Fanuc KAREL source: kt00178.KL

-- PROVISIONAL review KL for V1013-1; original PC SHA256 d3c23c733d1c245ba2e05406a3f4e00b66a2d6837c5a015371c1f33c9eca1489
-- Incomplete behavior may be omitted. Consult companion uncertainty JSON. Do not deploy.
PROGRAM KT00178
%NOLOCKGROUP
VAR
  I2 : INTEGER
  OUT : REAL
-- UNRESOLVED_DECL Y1 type=002018
BEGIN
  -- UNRESOLVED_PC offsets 5-19; opcodes 2E,22,9D,33,B2
  -- UNRESOLVED_PC offsets 24-35; opcodes 2E,23
  -- UNRESOLVED_PC offsets 40-63; opcodes 22,9D,33,B1,21,56,64,23
  -- UNRESOLVED_PC offsets 68-72; opcodes 7F
END KT00178
